% RSLogix 500 project PLC BASED WASHING MACHINE.RSS, saved by version 8.30.00.16 %
PROJECT "UNTITLED"    % processor: Bul.1763 MicroLogix 1100 Series B %

PROGRAM FILES
  LAD 2   21 rungs

DATA FILES
  O0 OUTPUT  4 elements
  I1 INPUT  6 elements
  S2 STATUS  66 elements
  B3 BINARY  1 elements
  T4 TIMER  8 elements
  C5 COUNTER  1 elements
  R6 CONTROL  1 elements
  N7 INTEGER  1 elements
  F8 FLOAT  1 elements

LADDER 2
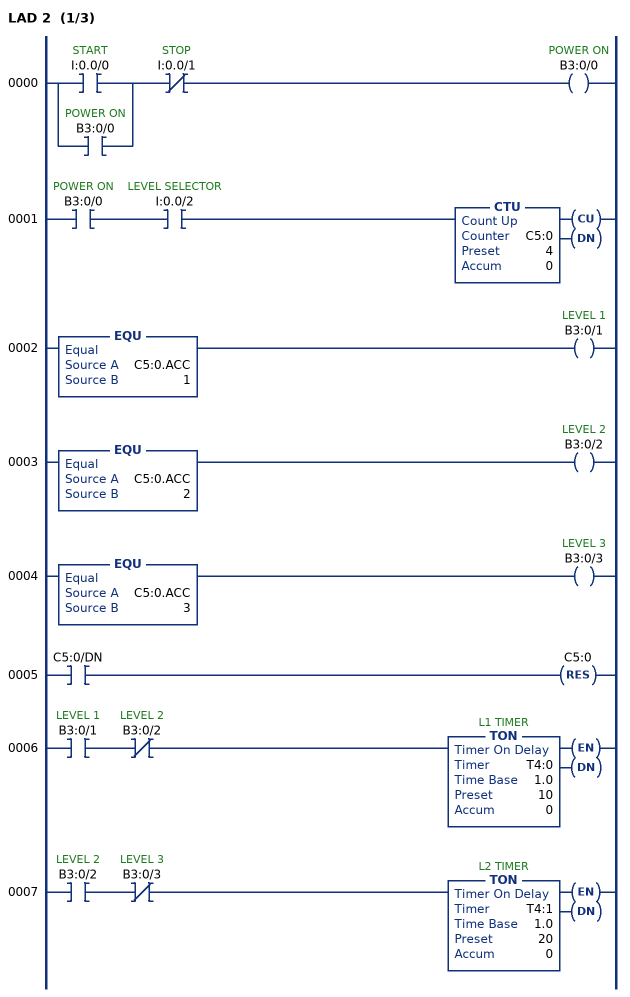
% Rung: 0 %
SOR BST XIC I:0.0/0 NXB XIC B3:0/0 BND XIO I:0.0/1 OTE B3:0/0 EOR
%   I:0.0/0  "START" %
%   B3:0/0  "POWER ON" %
%   I:0.0/1  "STOP" %
% Rung: 1 %
SOR XIC B3:0/0 XIC I:0.0/2 CTU C5:0 4 0 EOR
%   B3:0/0  "POWER ON" %
%   I:0.0/2  "LEVEL SELECTOR" %
% Rung: 2 %
SOR EQU C5:0.ACC 1 OTE B3:0/1 EOR
%   B3:0/1  "LEVEL 1" %
% Rung: 3 %
SOR EQU C5:0.ACC 2 OTE B3:0/2 EOR
%   B3:0/2  "LEVEL 2" %
% Rung: 4 %
SOR EQU C5:0.ACC 3 OTE B3:0/3 EOR
%   B3:0/3  "LEVEL 3" %
% Rung: 5 %
SOR XIC C5:0/DN RES C5:0 EOR
% Rung: 6 %
SOR XIC B3:0/1 XIO B3:0/2 TON T4:0 1.0 10 0 EOR
%   B3:0/1  "LEVEL 1" %
%   B3:0/2  "LEVEL 2" %
%   T4:0  "L1 TIMER" %
% Rung: 7 %
SOR XIC B3:0/2 XIO B3:0/3 TON T4:1 1.0 20 0 EOR
%   B3:0/2  "LEVEL 2" %
%   B3:0/3  "LEVEL 3" %
%   T4:1  "L2 TIMER" %

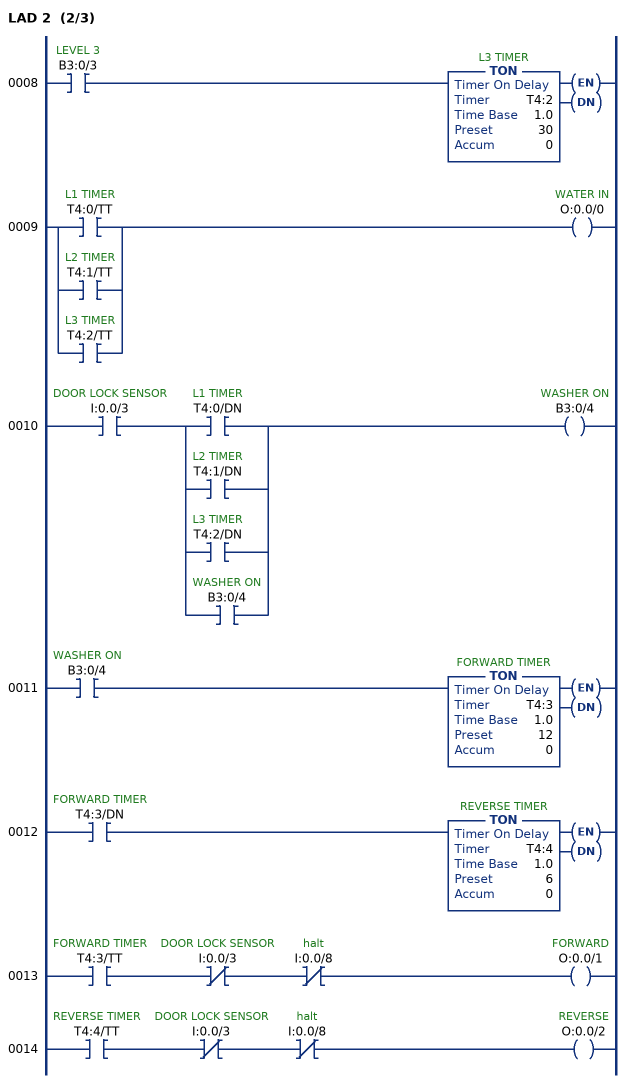
% Rung: 8 %
SOR XIC B3:0/3 TON T4:2 1.0 30 0 EOR
%   B3:0/3  "LEVEL 3" %
%   T4:2  "L3 TIMER" %
% Rung: 9 %
SOR BST XIC T4:0/TT NXB XIC T4:1/TT NXB XIC T4:2/TT BND OTE O:0.0/0 EOR
%   T4:0  "L1 TIMER" %
%   T4:1  "L2 TIMER" %
%   T4:2  "L3 TIMER" %
%   O:0.0/0  "WATER IN" %
% Rung: 10 %
SOR XIC I:0.0/3 BST XIC T4:0/DN NXB XIC T4:1/DN NXB XIC T4:2/DN NXB XIC B3:0/4 BND OTE B3:0/4 EOR
%   I:0.0/3  "DOOR LOCK SENSOR" %
%   T4:0  "L1 TIMER" %
%   T4:1  "L2 TIMER" %
%   T4:2  "L3 TIMER" %
%   B3:0/4  "WASHER ON" %
% Rung: 11 %
SOR XIC B3:0/4 TON T4:3 1.0 12 0 EOR
%   B3:0/4  "WASHER ON" %
%   T4:3  "FORWARD TIMER" %
% Rung: 12 %
SOR XIC T4:3/DN TON T4:4 1.0 6 0 EOR
%   T4:3  "FORWARD TIMER" %
%   T4:4  "REVERSE TIMER" %
% Rung: 13 %
SOR XIC T4:3/TT XIO I:0.0/3 XIO I:0.0/8 OTE O:0.0/1 EOR
%   T4:3  "FORWARD TIMER" %
%   I:0.0/3  "DOOR LOCK SENSOR" %
%   I:0.0/8  "halt" %
%   O:0.0/1  "FORWARD" %
% Rung: 14 %
SOR XIC T4:4/TT XIO I:0.0/3 XIO I:0.0/8 OTE O:0.0/2 EOR
%   T4:4  "REVERSE TIMER" %
%   I:0.0/3  "DOOR LOCK SENSOR" %
%   I:0.0/8  "halt" %
%   O:0.0/2  "REVERSE" %

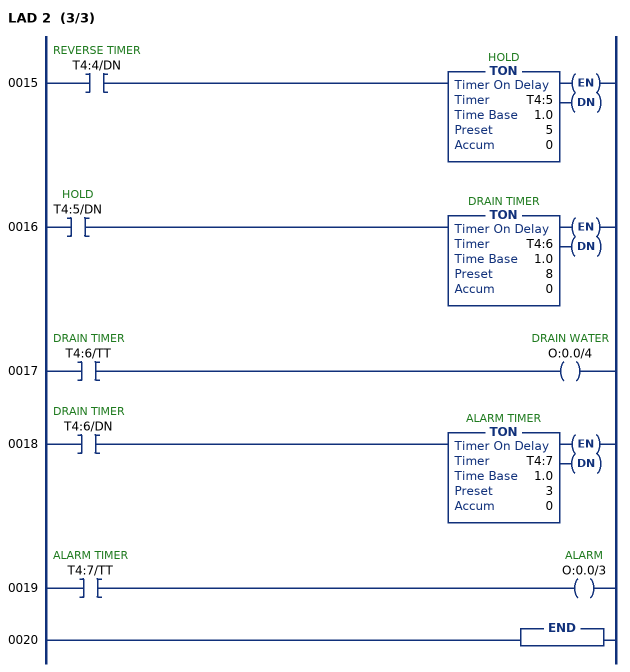
% Rung: 15 %
SOR XIC T4:4/DN TON T4:5 1.0 5 0 EOR
%   T4:4  "REVERSE TIMER" %
%   T4:5  "HOLD" %
% Rung: 16 %
SOR XIC T4:5/DN TON T4:6 1.0 8 0 EOR
%   T4:5  "HOLD" %
%   T4:6  "DRAIN TIMER" %
% Rung: 17 %
SOR XIC T4:6/TT OTE O:0.0/4 EOR
%   T4:6  "DRAIN TIMER" %
%   O:0.0/4  "DRAIN WATER" %
% Rung: 18 %
SOR XIC T4:6/DN TON T4:7 1.0 3 0 EOR
%   T4:6  "DRAIN TIMER" %
%   T4:7  "ALARM TIMER" %
% Rung: 19 %
SOR XIC T4:7/TT OTE O:0.0/3 EOR
%   T4:7  "ALARM TIMER" %
%   O:0.0/3  "ALARM" %
% Rung: 20 %
SOR END EOR

DATA TABLE (non-zero values as saved)
DATA T4
% .PRE .ACC %
% T4:0 % 10 0
% T4:1 % 20 0
% T4:2 % 30 0
% T4:3 % 12 0
% T4:4 % 6 0
% T4:5 % 5 0
% T4:6 % 8 0
% T4:7 % 3 0
DATA C5
% .PRE .ACC %
% C5:0 % 4 0
